(* PLC project steel-plant, Generated TextualNotationConverter 1.0 *)
(* stored: creationDateTime 2025-07-30T12:00:00, modificationDateTime 2025-01-30T12:00:00 *)

FUNCTION_BLOCK ANALOG_IN
  VAR_INPUT
    Name : STRING;
    Description : STRING;
    Raw_Signal : REAL;
    PV_High : REAL;
    PV_Low : REAL;
    Scaling_Slope : REAL;
    Scaling_Offset : REAL;
    Alarm_Enable : BOOL;
  END_VAR
  VAR_OUTPUT
    PV : REAL;
    High_Alarm : BOOL;
    Low_Alarm : BOOL;
    General_Fault : BOOL;
  END_VAR

            
          
END_FUNCTION_BLOCK

FUNCTION_BLOCK PID_BASIC
  VAR_INPUT
    Name : STRING;
    Description : STRING;
    AUTO : BOOL;
    PV : REAL;
    SP : REAL;
    MV_MIN : REAL;
    MV_MAX : REAL;
    X0 : REAL;
    KP : REAL;
    TR : REAL;
    TD : REAL;
    PV_High : REAL;
    PV_Low : REAL;
    Deviation_Limit : REAL;
    Inhibit : BOOL;
  END_VAR
  VAR_OUTPUT
    PV_High_Alarm : BOOL;
    PV_Low_Alarm : BOOL;
    Deviation_Alarm : BOOL;
    XOUT : REAL;
  END_VAR

            
          
END_FUNCTION_BLOCK

FUNCTION_BLOCK RATIO_CONTROL
  VAR_INPUT
    Name : STRING;
    Description : STRING;
    Auto : BOOL;
    PrimaryPV : REAL;
    SecondaryPV : REAL;
    RatioSP : REAL;
    Bias : REAL;
    TrimKp : REAL;
    TrimTi : STRING;
    MV_MIN : REAL;
    MV_MAX : REAL;
    ManOut : REAL;
    Inhibit : BOOL;
  END_VAR
  VAR_OUTPUT
    SlaveSP : REAL;
    ActiveRatio : REAL;
    RatioErr : REAL;
  END_VAR

            
          
END_FUNCTION_BLOCK

FUNCTION_BLOCK VALVE_ELECTRIC
  VAR_INPUT
    Name : STRING;
    Description : STRING;
    Control_Signal : REAL;
    Manual_Mode : BOOL;
    Manual_Position : REAL;
    Open_Limit : REAL;
    Close_Limit : REAL;
    Timeout : STRING;
    Inhibit : BOOL;
  END_VAR
  VAR_OUTPUT
    Valve_Position : REAL;
    Feedback_Pos : REAL;
    Valve_Moving : BOOL;
    Position_Error : BOOL;
    Alarm : BOOL;
  END_VAR

            
          
END_FUNCTION_BLOCK

PROGRAM Section2
  VAR
    FT101_WildFlow_PV : REAL;
    FT102_FluxFlow_PV : REAL;
    TIT101_Temperature_PV : REAL;
    FFIC103_FluxFlow_SP : REAL;
  END_VAR
  VAR
    FT-101 : ANALOG_IN;
    FT-102 : ANALOG_IN;
    TIT-101 : ANALOG_IN;
    FFIC-103 : RATIO_CONTROL;
    FIC-102 : PID_BASIC;
    FV-102 : VALVE_ELECTRIC;
  END_VAR
  VAR  (* added by the conversion: wires and edge detectors of the diagram *)
    _GT1_OUT : BOOL;
    _OR2_OUT : BOOL;
  END_VAR

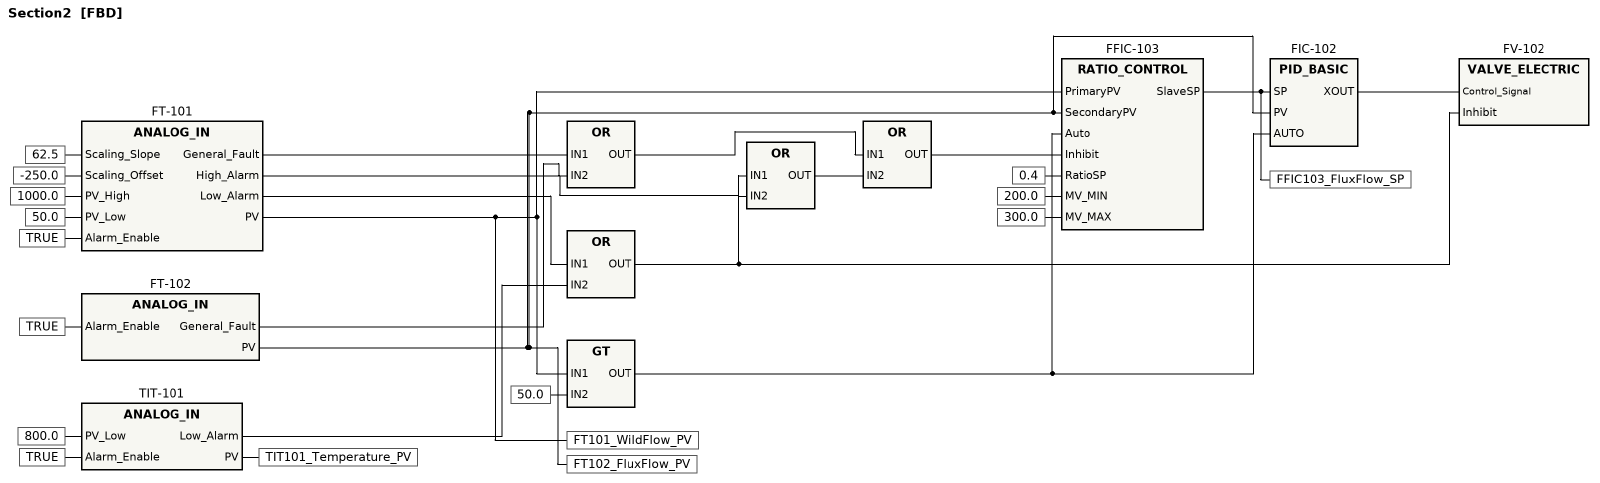
(* FBD diagram, written out as Structured Text *)
FT-101(Scaling_Slope := 62.5, Scaling_Offset := -250.0, PV_High := 1000.0, PV_Low := 50.0, Alarm_Enable := TRUE);
FT-102(Alarm_Enable := TRUE);
_GT1_OUT := FT-101.PV > 50.0;
TIT-101(PV_Low := 800.0, Alarm_Enable := TRUE);
_OR2_OUT := FT-101.Low_Alarm OR TIT-101.Low_Alarm;
FFIC-103(PrimaryPV := FT-101.PV, SecondaryPV := FT-102.PV, Auto := _GT1_OUT, Inhibit := FT-101.General_Fault OR FT-102.General_Fault OR FT-101.High_Alarm OR _OR2_OUT, RatioSP := 0.4, MV_MIN := 200.0, MV_MAX := 300.0);
FFIC103_FluxFlow_SP := FFIC-103.SlaveSP;
FT101_WildFlow_PV := FT-101.PV;
FT102_FluxFlow_PV := FT-102.PV;
TIT101_Temperature_PV := TIT-101.PV;
FIC-102(SP := FFIC-103.SlaveSP, PV := FT-102.PV, AUTO := _GT1_OUT);
FV-102(Control_Signal := FIC-102.XOUT, Inhibit := _OR2_OUT);
END_PROGRAM

FUNCTION_BLOCK BOOL_IN
  VAR_INPUT
    Name : STRING;
    Description : STRING;
    Bool_In : BOOL;
    Alarm_OnTrue : BOOL;
    Alarm_OnFalse : BOOL;
    Latch_Enable : BOOL;
    Reset_Latch : BOOL;
  END_VAR
  VAR_OUTPUT
    Bool_Out : BOOL;
    Alarm_Active : BOOL;
    Latched_Status : BOOL;
  END_VAR

            
          
END_FUNCTION_BLOCK

FUNCTION_BLOCK DIGITAL_IN
  VAR_INPUT
    Name : STRING;
    Description : STRING;
    DI_Raw : BOOL;
    DebounceTime : STRING;
    EnableAlarm : BOOL;
  END_VAR
  VAR_OUTPUT
    DI_Out : BOOL;
    Fault_State : BOOL;
  END_VAR

            
          
END_FUNCTION_BLOCK

FUNCTION_BLOCK DUTY_STANDBY
  VAR_INPUT
    Name : STRING;
    Description : STRING;
    Enable : BOOL;
    StartRequest : BOOL;
    AlternateEnable : BOOL;
    ForcePumpA : BOOL;
    ForcePumpB : BOOL;
    DutyElapsed : BOOL;
    MinRunElapsed : BOOL;
    SwitchoverDelayElapsed : BOOL;
    StartTimeoutElapsed : BOOL;
    PumpA_RunFB : BOOL;
    PumpB_RunFB : BOOL;
    PumpA_Fault : BOOL;
    PumpB_Fault : BOOL;
    Reset : BOOL;
    Inhibit : BOOL;
  END_VAR
  VAR_OUTPUT
    CmdPumpA : BOOL;
    CmdPumpB : BOOL;
    ActiveIsA : BOOL;
    SwitchedDueToDuty : BOOL;
    SwitchedDueToFailure : BOOL;
    Alarm_FailedStart_A : BOOL;
    Alarm_FailedStart_B : BOOL;
    Alarm_NoAvailablePump : BOOL;
  END_VAR

            
          
END_FUNCTION_BLOCK

FUNCTION_BLOCK MOTOR_2SPD
  VAR_INPUT
    Name : STRING;
    Description : STRING;
    Start_Cmd : BOOL;
    Stop_Cmd : BOOL;
    Speed_High_Cmd : BOOL;
    Speed_Low_Cmd : BOOL;
    Inhibit : BOOL;
  END_VAR
  VAR_OUTPUT
    Motor_Start_Out : BOOL;
    FB_Running : BOOL;
    FB_Trip : BOOL;
    FB_HighSpeed : BOOL;
    FB_LowSpeed : BOOL;
    Alarm_Speed_Error : BOOL;
  END_VAR

            
          
END_FUNCTION_BLOCK

FUNCTION_BLOCK MOTOR_ON_OFF
  VAR_INPUT
    Name : STRING;
    Description : STRING;
    Start_Cmd : BOOL;
    Stop_Cmd : BOOL;
    Start_Delay : STRING;
    MinRunTime : STRING;
    Inhibit : BOOL;
  END_VAR
  VAR_OUTPUT
    Motor_Start_Out : BOOL;
    FB_Running : BOOL;
    FB_Trip : BOOL;
    Alarm_Start_Fail : BOOL;
    Alarm_Stop_Fail : BOOL;
  END_VAR

            
          
END_FUNCTION_BLOCK

FUNCTION_BLOCK MOTOR_VSD
  VAR_INPUT
    Name : STRING;
    Description : STRING;
    Start_Cmd : BOOL;
    Stop_Cmd : BOOL;
    Speed_SP : REAL;
    Accel_Ramp : STRING;
    Decel_Ramp : STRING;
    Inhibit : BOOL;
  END_VAR
  VAR_OUTPUT
    Speed_Out : REAL;
    FB_Running : BOOL;
    FB_Fault : BOOL;
    FB_Ready : BOOL;
    FB_ActualSpeed : REAL;
    Alarm_Speed_Deviation : BOOL;
    Alarm_Comm_Fail : BOOL;
  END_VAR

            
          
END_FUNCTION_BLOCK

FUNCTION_BLOCK SPLIT_RANGE
  VAR_INPUT
    Name : STRING;
    Description : STRING;
    IN : REAL;
    Split_Point : REAL;
    Output1_Start : REAL;
    Output1_End : REAL;
    Output2_Start : REAL;
    Output2_End : REAL;
  END_VAR
  VAR_OUTPUT
    OUT1 : REAL;
    OUT2 : REAL;
  END_VAR

            
          
END_FUNCTION_BLOCK

FUNCTION_BLOCK VALVE_ON_OFF
  VAR_INPUT
    Name : STRING;
    Description : STRING;
    Open_Cmd : BOOL;
    Close_Cmd : BOOL;
    Timeout : STRING;
    Inhibit : BOOL;
  END_VAR
  VAR_OUTPUT
    FB_Opened : BOOL;
    FB_Closed : BOOL;
    Valve_Open_Out : BOOL;
    Valve_Close_Out : BOOL;
    Alarm_Position_Error : BOOL;
    Alarm_General : BOOL;
  END_VAR

            
          
END_FUNCTION_BLOCK

FUNCTION_BLOCK VOTING_ANALOG
  VAR_INPUT
    Name : STRING;
    Description : STRING;
    Input1 : REAL;
    Input2 : REAL;
    Input3 : REAL;
    Deviation_Limit : REAL;
    Voting_Scheme : STRING;
    EnableAlarm : BOOL;
    Inhibit : BOOL;
  END_VAR
  VAR_OUTPUT
    Voted_Output : REAL;
    Sensor1_Fault : BOOL;
    Sensor2_Fault : BOOL;
    Sensor3_Fault : BOOL;
    Alarm_Voting_Error : BOOL;
    Healthy_Sensors_Count : INT;
  END_VAR

            
          
END_FUNCTION_BLOCK

PROGRAM Section3
  VAR
    PT_201_VOTE_PV : REAL;
    TT_201_VOTE_PV : REAL;
  END_VAR
  VAR
    PT-201A : ANALOG_IN;
    PT-201B : ANALOG_IN;
    PT-201C : ANALOG_IN;
    TT-201A : ANALOG_IN;
    TT-201B : ANALOG_IN;
    TT-201C : ANALOG_IN;
    PT-201_VOTE : VOTING_ANALOG;
    TT-201_VOTE : VOTING_ANALOG;
    P-201 : MOTOR_ON_OFF;
    MO-201 : DIGITAL_IN;
    MO-202 : DIGITAL_IN;
    I-201 : BOOL_IN;
    I-202 : BOOL_IN;
    SI-201 : BOOL_IN;
    SI-202 : BOOL_IN;
  END_VAR
  VAR  (* added by the conversion: wires and edge detectors of the diagram *)
    _OR37_OUT : BOOL;
  END_VAR

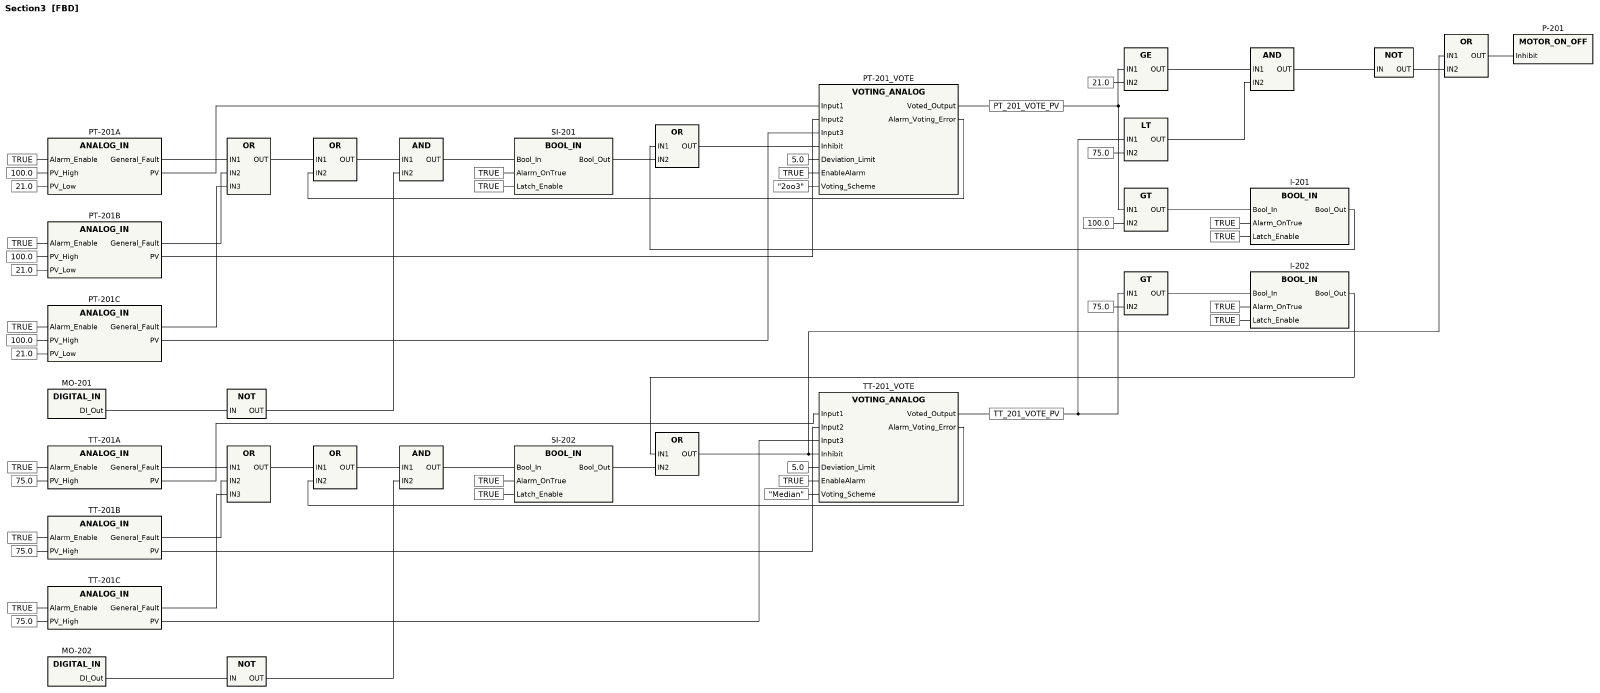
(* FBD diagram, written out as Structured Text *)
PT-201A(Alarm_Enable := TRUE, PV_High := 100.0, PV_Low := 21.0);
PT-201B(Alarm_Enable := TRUE, PV_High := 100.0, PV_Low := 21.0);
PT-201C(Alarm_Enable := TRUE, PV_High := 100.0, PV_Low := 21.0);
I-201(Bool_In := PT-201_VOTE.Voted_Output > 100.0, Alarm_OnTrue := TRUE, Latch_Enable := TRUE);
MO-201();
SI-201(Bool_In := (PT-201A.General_Fault OR PT-201B.General_Fault OR PT-201C.General_Fault OR PT-201_VOTE.Alarm_Voting_Error) AND NOT MO-201.DI_Out, Alarm_OnTrue := TRUE, Latch_Enable := TRUE);
PT-201_VOTE(Input1 := PT-201A.PV, Input2 := PT-201B.PV, Input3 := PT-201C.PV, Inhibit := I-201.Bool_Out OR SI-201.Bool_Out, Deviation_Limit := 5.0, EnableAlarm := TRUE, Voting_Scheme := "2oo3");
PT_201_VOTE_PV := PT-201_VOTE.Voted_Output;
TT-201A(Alarm_Enable := TRUE, PV_High := 75.0);
TT-201B(Alarm_Enable := TRUE, PV_High := 75.0);
TT-201C(Alarm_Enable := TRUE, PV_High := 75.0);
I-202(Bool_In := TT-201_VOTE.Voted_Output > 75.0, Alarm_OnTrue := TRUE, Latch_Enable := TRUE);
MO-202();
SI-202(Bool_In := (TT-201A.General_Fault OR TT-201B.General_Fault OR TT-201C.General_Fault OR TT-201_VOTE.Alarm_Voting_Error) AND NOT MO-202.DI_Out, Alarm_OnTrue := TRUE, Latch_Enable := TRUE);
_OR37_OUT := I-202.Bool_Out OR SI-202.Bool_Out;
TT-201_VOTE(Input1 := TT-201A.PV, Input2 := TT-201B.PV, Input3 := TT-201C.PV, Inhibit := _OR37_OUT, Deviation_Limit := 5.0, EnableAlarm := TRUE, Voting_Scheme := "Median");
TT_201_VOTE_PV := TT-201_VOTE.Voted_Output;
P-201(Inhibit := _OR37_OUT OR NOT (PT-201_VOTE.Voted_Output >= 21.0 AND TT-201_VOTE.Voted_Output < 75.0));
END_PROGRAM

PROGRAM Section4
  VAR
    FT_301_CoalFlow_PV : REAL;
    FT_302_AirFlow_PV : REAL;
    PT_301_Pressure_PV : REAL;
    TT_301_Temperature_PV : REAL;
    FIC_302_HotBlastAir_SP_FromRatio : REAL;
    Ratio_Bias : REAL;
  END_VAR
  VAR
    FT-301 : ANALOG_IN;
    PT-301 : ANALOG_IN;
    TT-301 : ANALOG_IN;
    FT-302 : ANALOG_IN;
    FFIC-303 : RATIO_CONTROL;
    FIC-302 : PID_BASIC;
    FV-302 : VALVE_ELECTRIC;
  END_VAR
  VAR  (* added by the conversion: wires and edge detectors of the diagram *)
    _OR95_OUT : BOOL;
    _OR96_OUT : BOOL;
  END_VAR

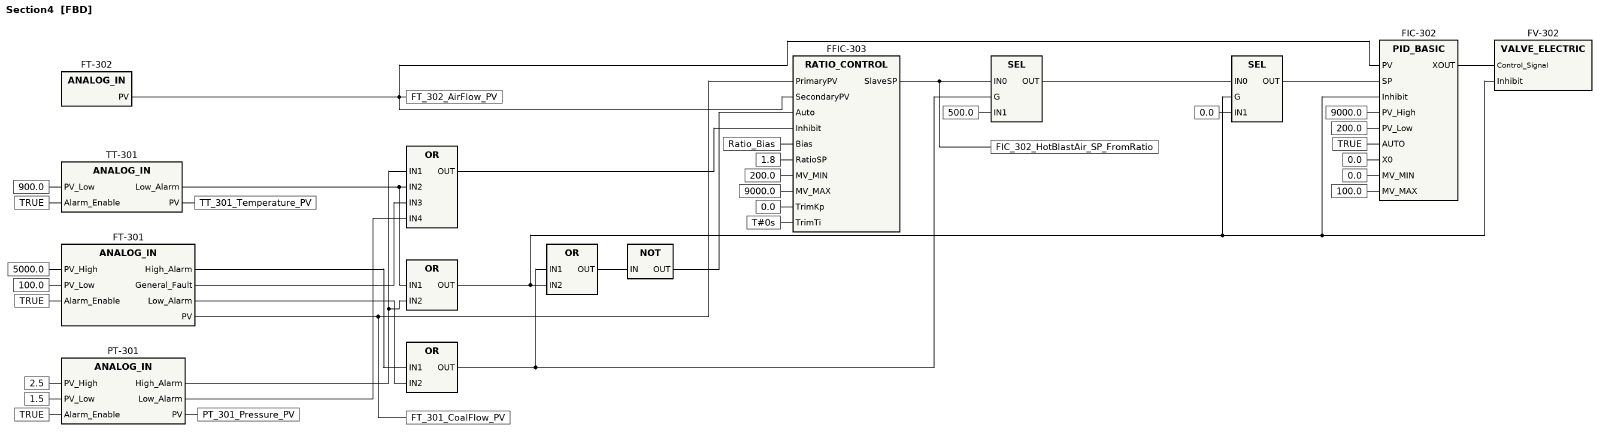
(* FBD diagram, written out as Structured Text *)
FT-301(PV_High := 5000.0, PV_Low := 100.0, Alarm_Enable := TRUE);
FT-302();
_OR95_OUT := FT-301.High_Alarm OR FT-301.Low_Alarm;
TT-301(PV_Low := 900.0, Alarm_Enable := TRUE);
PT-301(PV_High := 2.5, PV_Low := 1.5, Alarm_Enable := TRUE);
_OR96_OUT := TT-301.Low_Alarm OR PT-301.High_Alarm;
FFIC-303(PrimaryPV := FT-301.PV, SecondaryPV := FT-302.PV, Auto := NOT (_OR95_OUT OR _OR96_OUT), Inhibit := PT-301.High_Alarm OR TT-301.Low_Alarm OR FT-301.General_Fault OR PT-301.Low_Alarm, Bias := Ratio_Bias, RatioSP := 1.8, MV_MIN := 200.0, MV_MAX := 9000.0, TrimKp := 0.0, TrimTi := T#0s);
FIC_302_HotBlastAir_SP_FromRatio := FFIC-303.SlaveSP;
FT_301_CoalFlow_PV := FT-301.PV;
FT_302_AirFlow_PV := FT-302.PV;
PT_301_Pressure_PV := PT-301.PV;
TT_301_Temperature_PV := TT-301.PV;
FIC-302(PV := FT-302.PV, SP := SEL(SEL(FFIC-303.SlaveSP, _OR95_OUT, 500.0), _OR96_OUT, 0.0), Inhibit := _OR96_OUT, PV_High := 9000.0, PV_Low := 200.0, AUTO := TRUE, X0 := 0.0, MV_MIN := 0.0, MV_MAX := 100.0);
FV-302(Control_Signal := FIC-302.XOUT, Inhibit := _OR96_OUT);
END_PROGRAM

PROGRAM Section5
  VAR
    TT_401_V_Temp_PV : REAL;
    PT_401_V_Pressure_PV : REAL;
    FT_401_Flow_PV : REAL;
  END_VAR
  VAR
    FT-401 : ANALOG_IN;
    PT-401A : ANALOG_IN;
    PT-401B : ANALOG_IN;
    PT-401C : ANALOG_IN;
    TT-401 : ANALOG_IN;
    TT-401A : ANALOG_IN;
    TT-401B : ANALOG_IN;
    TT-401C : ANALOG_IN;
    TT-401-V : VOTING_ANALOG;
    PT-401-V : VOTING_ANALOG;
    BOF-401_TempControl : PID_BASIC;
    BOF-402 : VALVE_ELECTRIC;
    I-401 : BOOL_IN;
    MA-401 : BOOL_IN;
    DA-401 : BOOL_IN;
    FA-401 : BOOL_IN;
  END_VAR
  VAR  (* added by the conversion: wires and edge detectors of the diagram *)
    _AND143_OUT : BOOL;
    _AND144_OUT : BOOL;
    _AND145_OUT : BOOL;
  END_VAR

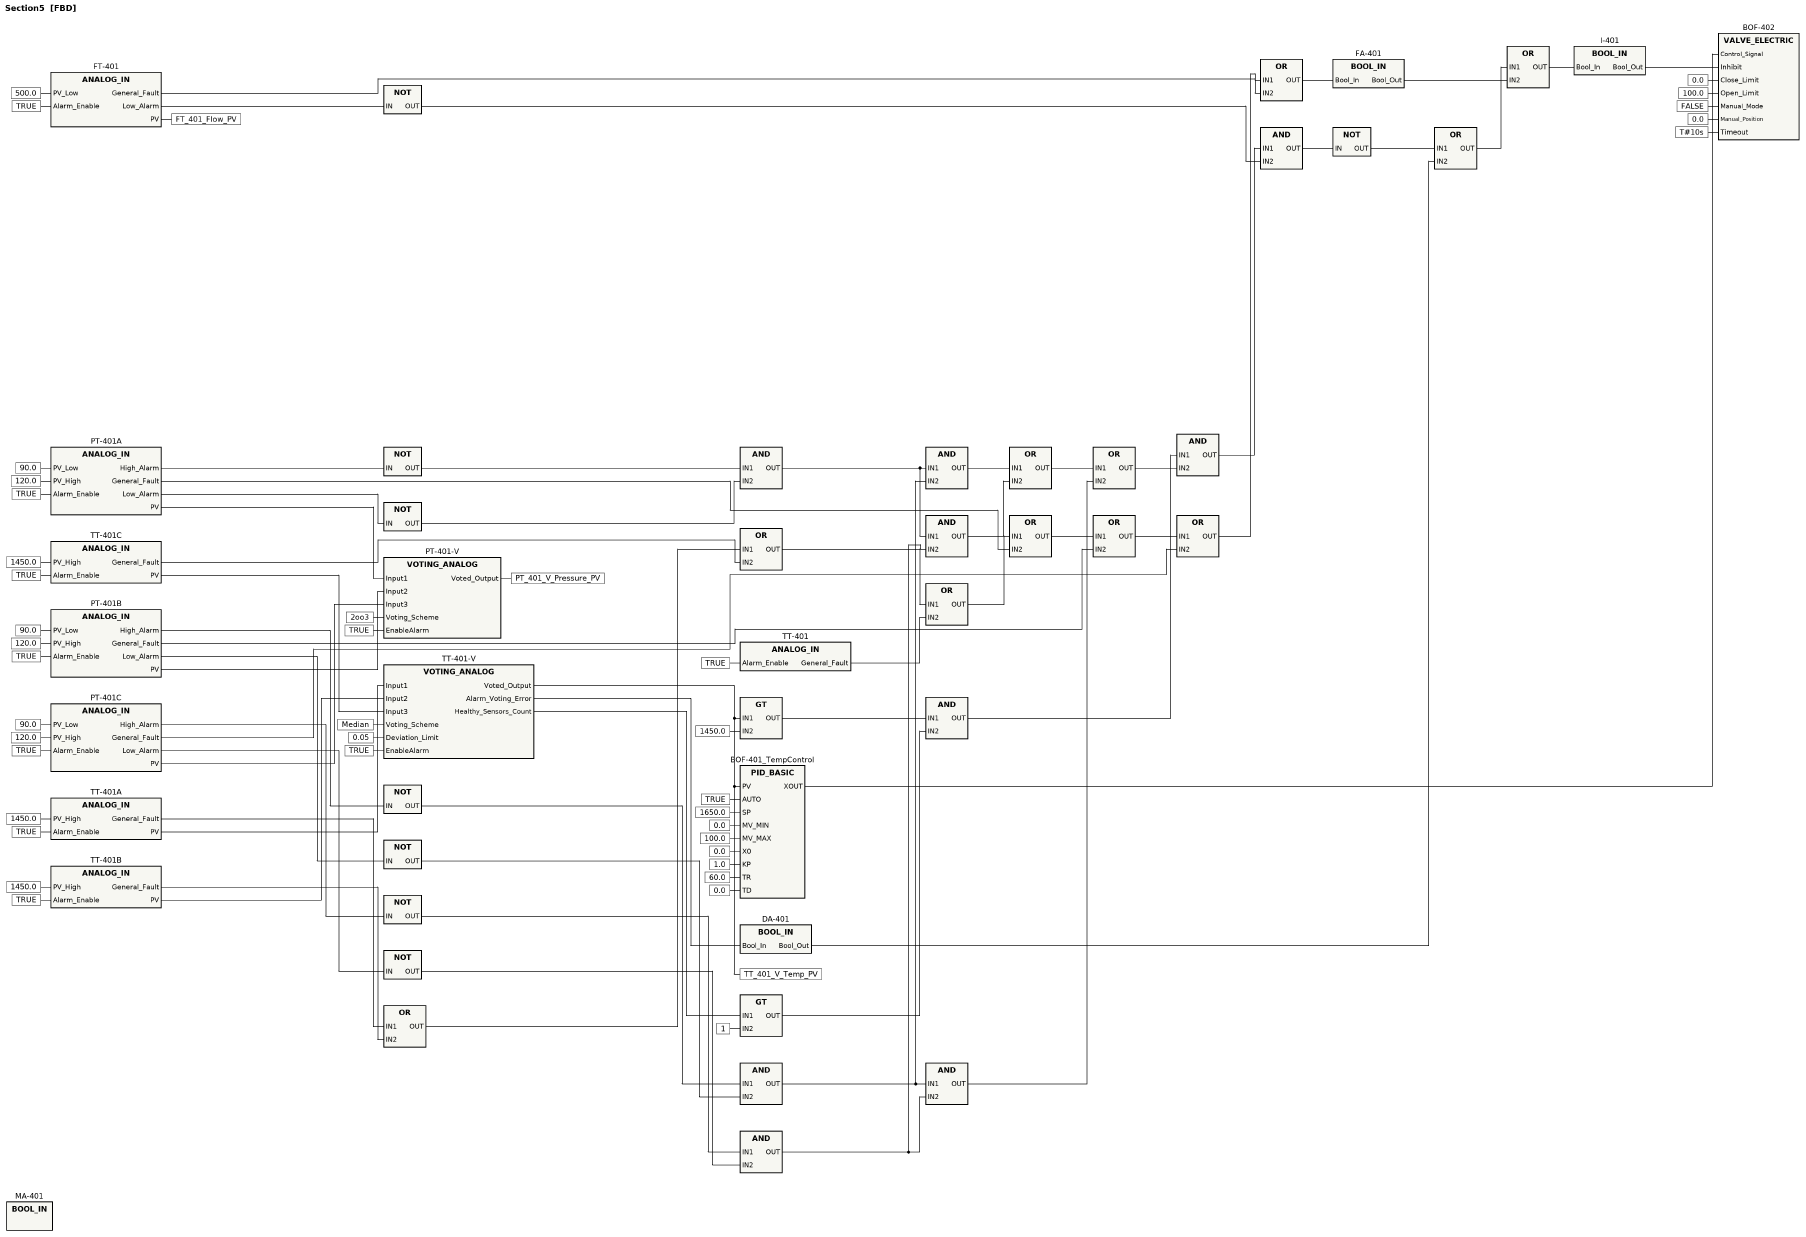
(* FBD diagram, written out as Structured Text *)
FT-401(PV_Low := 500.0, Alarm_Enable := TRUE);
FT_401_Flow_PV := FT-401.PV;
PT-401A(PV_Low := 90.0, PV_High := 120.0, Alarm_Enable := TRUE);
PT-401B(PV_Low := 90.0, PV_High := 120.0, Alarm_Enable := TRUE);
PT-401C(PV_Low := 90.0, PV_High := 120.0, Alarm_Enable := TRUE);
PT-401-V(Input1 := PT-401A.PV, Input2 := PT-401B.PV, Input3 := PT-401C.PV, Voting_Scheme := 2oo3, EnableAlarm := TRUE);
PT_401_V_Pressure_PV := PT-401-V.Voted_Output;
TT-401A(PV_High := 1450.0, Alarm_Enable := TRUE);
TT-401B(PV_High := 1450.0, Alarm_Enable := TRUE);
TT-401C(PV_High := 1450.0, Alarm_Enable := TRUE);
TT-401-V(Input1 := TT-401A.PV, Input2 := TT-401B.PV, Input3 := TT-401C.PV, Voting_Scheme := Median, Deviation_Limit := 0.05, EnableAlarm := TRUE);
TT_401_V_Temp_PV := TT-401-V.Voted_Output;
_AND143_OUT := NOT PT-401A.High_Alarm AND NOT PT-401A.Low_Alarm;
_AND144_OUT := NOT PT-401B.High_Alarm AND NOT PT-401B.Low_Alarm;
_AND145_OUT := NOT PT-401C.High_Alarm AND NOT PT-401C.Low_Alarm;
TT-401(Alarm_Enable := TRUE);
DA-401(Bool_In := TT-401-V.Alarm_Voting_Error);
FA-401(Bool_In := TT-401A.General_Fault OR TT-401B.General_Fault OR TT-401C.General_Fault OR TT-401.General_Fault OR PT-401A.General_Fault OR PT-401B.General_Fault OR PT-401C.General_Fault OR FT-401.General_Fault);
BOF-401_TempControl(PV := TT-401-V.Voted_Output, AUTO := TRUE, SP := 1650.0, MV_MIN := 0.0, MV_MAX := 100.0, X0 := 0.0, KP := 1.0, TR := 60.0, TD := 0.0);
I-401(Bool_In := NOT (TT-401-V.Voted_Output > 1450.0 AND TT-401-V.Healthy_Sensors_Count > 1 AND (_AND143_OUT AND _AND144_OUT OR _AND143_OUT AND _AND145_OUT OR _AND144_OUT AND _AND145_OUT) AND NOT FT-401.Low_Alarm) OR DA-401.Bool_Out OR FA-401.Bool_Out);
BOF-402(Control_Signal := BOF-401_TempControl.XOUT, Inhibit := I-401.Bool_Out, Close_Limit := 0.0, Open_Limit := 100.0, Manual_Mode := FALSE, Manual_Position := 0.0, Timeout := T#10s);
MA-401();
END_PROGRAM

PROGRAM Section6
  VAR
    PT_501_Pressure_PV : REAL;
    TT_501_Temperature_PV : REAL;
    TT_501_MV : REAL;
    SM_501_EA_POS : REAL;
    SM_501_EA_CMD : REAL;
  END_VAR
  VAR
    PT-501 : ANALOG_IN;
    TT-501 : ANALOG_IN;
    SM-501 : VALVE_ELECTRIC;
    TT-501_CTRL : PID_BASIC;
    SM-501.LID_POS : DIGITAL_IN;
    HeatingEnableDelay_TON : TON;
  END_VAR
  VAR  (* added by the conversion: wires and edge detectors of the diagram *)
    _OR223_OUT : BOOL;
  END_VAR

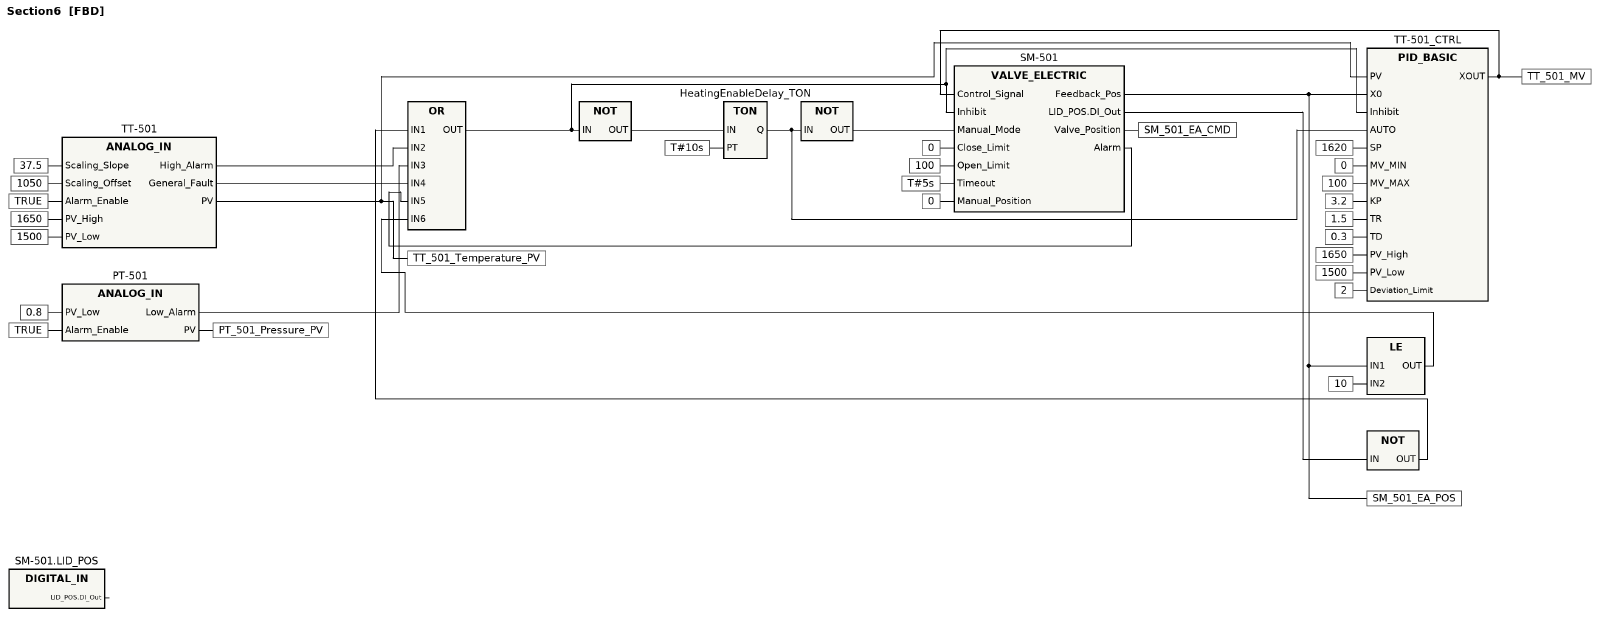
(* FBD diagram, written out as Structured Text *)
PT-501(PV_Low := 0.8, Alarm_Enable := TRUE);
PT_501_Pressure_PV := PT-501.PV;
TT-501(Scaling_Slope := 37.5, Scaling_Offset := 1050, Alarm_Enable := TRUE, PV_High := 1650, PV_Low := 1500);
_OR223_OUT := NOT SM-501.LID_POS.DI_Out OR TT-501.High_Alarm OR PT-501.Low_Alarm OR TT-501.General_Fault OR SM-501.Alarm OR SM-501.Feedback_Pos <= 10;
HeatingEnableDelay_TON(IN := NOT _OR223_OUT, PT := T#10s);
TT-501_CTRL(PV := TT-501.PV, X0 := SM-501.Feedback_Pos, Inhibit := _OR223_OUT, AUTO := HeatingEnableDelay_TON.Q, SP := 1620, MV_MIN := 0, MV_MAX := 100, KP := 3.2, TR := 1.5, TD := 0.3, PV_High := 1650, PV_Low := 1500, Deviation_Limit := 2);
SM-501(Control_Signal := TT-501_CTRL.XOUT, Inhibit := _OR223_OUT, Manual_Mode := NOT HeatingEnableDelay_TON.Q, Close_Limit := 0, Open_Limit := 100, Timeout := T#5s, Manual_Position := 0);
SM_501_EA_CMD := SM-501.Valve_Position;
SM_501_EA_POS := SM-501.Feedback_Pos;
TT_501_MV := TT-501_CTRL.XOUT;
TT_501_Temperature_PV := TT-501.PV;
SM-501.LID_POS();
END_PROGRAM

PROGRAM Section7
  VAR
    LIT101_MoldLevel_PV_mm : REAL;
    FT601_CoolingWaterFlow_PV_m3h : REAL;
    TT601_MoldTemp_PV_C : REAL;
    LIC101_ControllerOutput_Pct : REAL;
  END_VAR
  VAR
    LIT-101 : ANALOG_IN;
    FT-601 : ANALOG_IN;
    TT-601 : ANALOG_IN;
    LIC-101 : PID_BASIC;
    MV-101 : VALVE_ELECTRIC;
    ILK-FT-601-LOW : BOOL_IN;
    ILK-TT-601-HIGH : BOOL_IN;
    PERM-LIT-101-UNDER-250 : BOOL_IN;
    ILK-LIT-101-HIGH-HIGH-280 : BOOL_IN;
    ILK-LIT-101-FAULT : BOOL_IN;
  END_VAR
  VAR  (* added by the conversion: wires and edge detectors of the diagram *)
    _OR261_OUT : BOOL;
  END_VAR

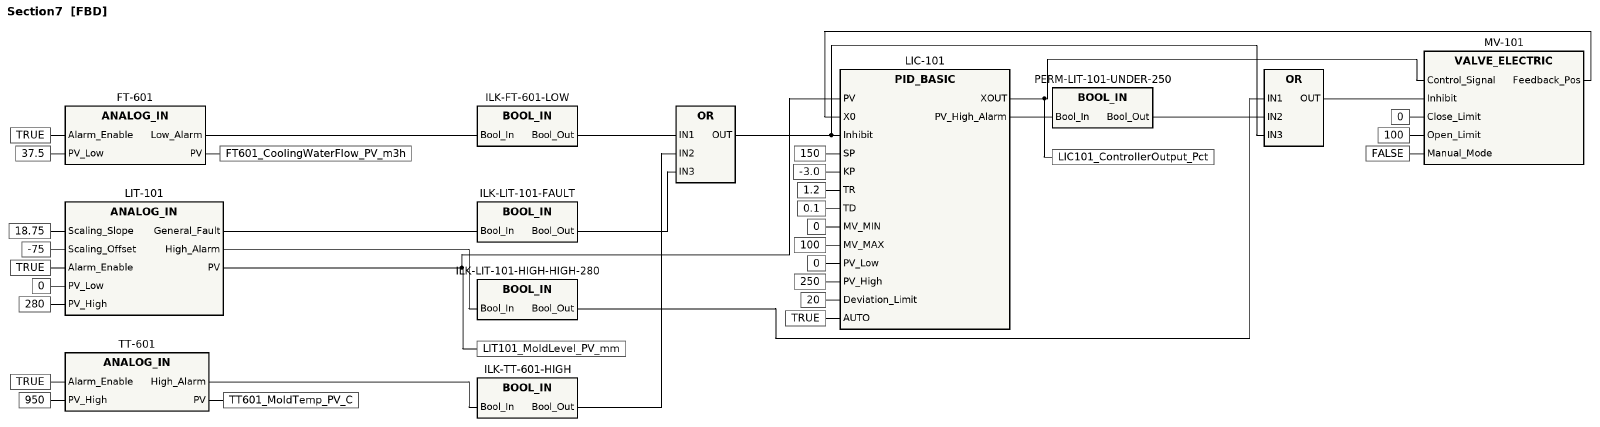
(* FBD diagram, written out as Structured Text *)
FT-601(Alarm_Enable := TRUE, PV_Low := 37.5);
FT601_CoolingWaterFlow_PV_m3h := FT-601.PV;
LIT-101(Scaling_Slope := 18.75, Scaling_Offset := -75, Alarm_Enable := TRUE, PV_Low := 0, PV_High := 280);
ILK-LIT-101-HIGH-HIGH-280(Bool_In := LIT-101.High_Alarm);
PERM-LIT-101-UNDER-250(Bool_In := LIC-101.PV_High_Alarm);
ILK-FT-601-LOW(Bool_In := FT-601.Low_Alarm);
TT-601(Alarm_Enable := TRUE, PV_High := 950);
ILK-TT-601-HIGH(Bool_In := TT-601.High_Alarm);
ILK-LIT-101-FAULT(Bool_In := LIT-101.General_Fault);
_OR261_OUT := ILK-FT-601-LOW.Bool_Out OR ILK-TT-601-HIGH.Bool_Out OR ILK-LIT-101-FAULT.Bool_Out;
MV-101(Control_Signal := LIC-101.XOUT, Inhibit := ILK-LIT-101-HIGH-HIGH-280.Bool_Out OR PERM-LIT-101-UNDER-250.Bool_Out OR _OR261_OUT, Close_Limit := 0, Open_Limit := 100, Manual_Mode := FALSE);
LIC-101(PV := LIT-101.PV, X0 := MV-101.Feedback_Pos, Inhibit := _OR261_OUT, SP := 150, KP := -3.0, TR := 1.2, TD := 0.1, MV_MIN := 0, MV_MAX := 100, PV_Low := 0, PV_High := 250, Deviation_Limit := 20, AUTO := TRUE);
LIC101_ControllerOutput_Pct := LIC-101.XOUT;
LIT101_MoldLevel_PV_mm := LIT-101.PV;
TT601_MoldTemp_PV_C := TT-601.PV;
END_PROGRAM

PROGRAM Section8
  VAR
    FT701_FuelFlow_PV : REAL;
    FT702_AirFlow_PV : REAL;
    TT701_FurnaceTemp_PV : REAL;
    FLT701_FuelTankLevel_PV : REAL;
    FT702_SP_Ratio : REAL;
    FFIC701_ActiveRatio : REAL;
    FFIC701_RatioError : REAL;
    BLS701_BurnerStatus : BOOL;
    BLS701_BurnerStatus_DI : BOOL;
    ALM701_RatioAlarm : BOOL;
    ALM702_FT701Fault : BOOL;
    ALM703_FT702Fault : BOOL;
    ALM704_HighTemp : BOOL;
  END_VAR
  VAR
    FT-701 : ANALOG_IN;
    FT-702 : ANALOG_IN;
    TT-701 : ANALOG_IN;
    FLT-701 : ANALOG_IN;
    FFIC-701 : RATIO_CONTROL;
    FIC-702 : PID_BASIC;
    FV-702 : VALVE_ELECTRIC;
    BLS-701 : BOOL_IN;
  END_VAR
  VAR  (* added by the conversion: wires and edge detectors of the diagram *)
    _NOT300_OUT : BOOL;
    _OR301_OUT : BOOL;
  END_VAR

(* FBD diagram, written out as Structured Text *)
FT-701(PV_High := 5000.0, PV_Low := 200.0, Alarm_Enable := TRUE);
FT-702(PV_High := 15000.0, PV_Low := 0.0, Alarm_Enable := TRUE);
TT-701(PV_High := 1200.0, PV_Low := 800.0, Alarm_Enable := TRUE);
BLS-701(Bool_In := BLS701_BurnerStatus_DI, Alarm_OnFalse := TRUE, Alarm_OnTrue := FALSE, Latch_Enable := FALSE);
_NOT300_OUT := NOT BLS-701.Bool_Out;
_OR301_OUT := FT-701.General_Fault OR FT-702.General_Fault;
FFIC-701(PrimaryPV := FT-701.PV, SecondaryPV := FT-702.PV, Auto := NOT TT-701.High_Alarm AND FT-701.PV >= 200.0 AND BLS-701.Bool_Out, Inhibit := _NOT300_OUT OR FT-701.Low_Alarm OR _OR301_OUT, MV_MIN := MULT(FT-701.PV, 8.0), MV_MAX := MULT(FT-701.PV, 12.0), ManOut := MULT(FT-701.PV, 8.0), RatioSP := 10.0, Bias := 0.0);
ALM701_RatioAlarm := FFIC-701.ActiveRatio > 8.0 OR FFIC-701.ActiveRatio > 12.0;
ALM702_FT701Fault := FT-701.General_Fault;
ALM703_FT702Fault := FT-702.General_Fault;
ALM704_HighTemp := TT-701.High_Alarm;
BLS701_BurnerStatus := BLS-701.Bool_Out;
FFIC701_ActiveRatio := FFIC-701.ActiveRatio;
FFIC701_RatioError := FFIC-701.RatioErr;
FLT-701();
FLT701_FuelTankLevel_PV := FLT-701.PV;
FT701_FuelFlow_PV := FT-701.PV;
FT702_AirFlow_PV := FT-702.PV;
FT702_SP_Ratio := FFIC-701.SlaveSP;
TT701_FurnaceTemp_PV := TT-701.PV;
FIC-702(SP := FFIC-701.SlaveSP, PV := FT-702.PV, Inhibit := _NOT300_OUT OR _OR301_OUT, AUTO := TRUE, MV_MIN := 0.0, MV_MAX := 100.0, PV_High := 15000.0, PV_Low := 0.0, KP := 1.5, TR := 10.0, TD := 0.5, Deviation_Limit := 5.0, X0 := 0.0);
FV-702(Control_Signal := FIC-702.XOUT, Inhibit := FT-701.Low_Alarm OR TT-701.Low_Alarm OR TT-701.High_Alarm OR _OR301_OUT, Manual_Mode := FALSE, Close_Limit := 0.0, Open_Limit := 100.0, Timeout := T#10s);
END_PROGRAM

PROGRAM Section9
  VAR
    FT801_Flow_PV : REAL;
    FT802_Flow_PV : REAL;
    PT801_Pressure_PV : REAL;
    FFIC801_AirFlow_SP : REAL;
    FFIC801_ActiveRatio : REAL;
    RatioHigh_Alarm : BOOL;
    RatioLow_Alarm : BOOL;
  END_VAR
  VAR
    AL-801 : ANALOG_IN;
    AL-802 : ANALOG_IN;
    AL-803 : ANALOG_IN;
    AL-804 : ANALOG_IN;
    FT-801 : ANALOG_IN;
    FT-802 : ANALOG_IN;
    PT-801 : ANALOG_IN;
    FFIC-801 : RATIO_CONTROL;
    FIC-802 : PID_BASIC;
    FV-802 : VALVE_ELECTRIC;
  END_VAR
  VAR  (* added by the conversion: wires and edge detectors of the diagram *)
    _GE372_OUT : BOOL;
    _OR373_OUT : BOOL;
    _OR375_OUT : BOOL;
  END_VAR

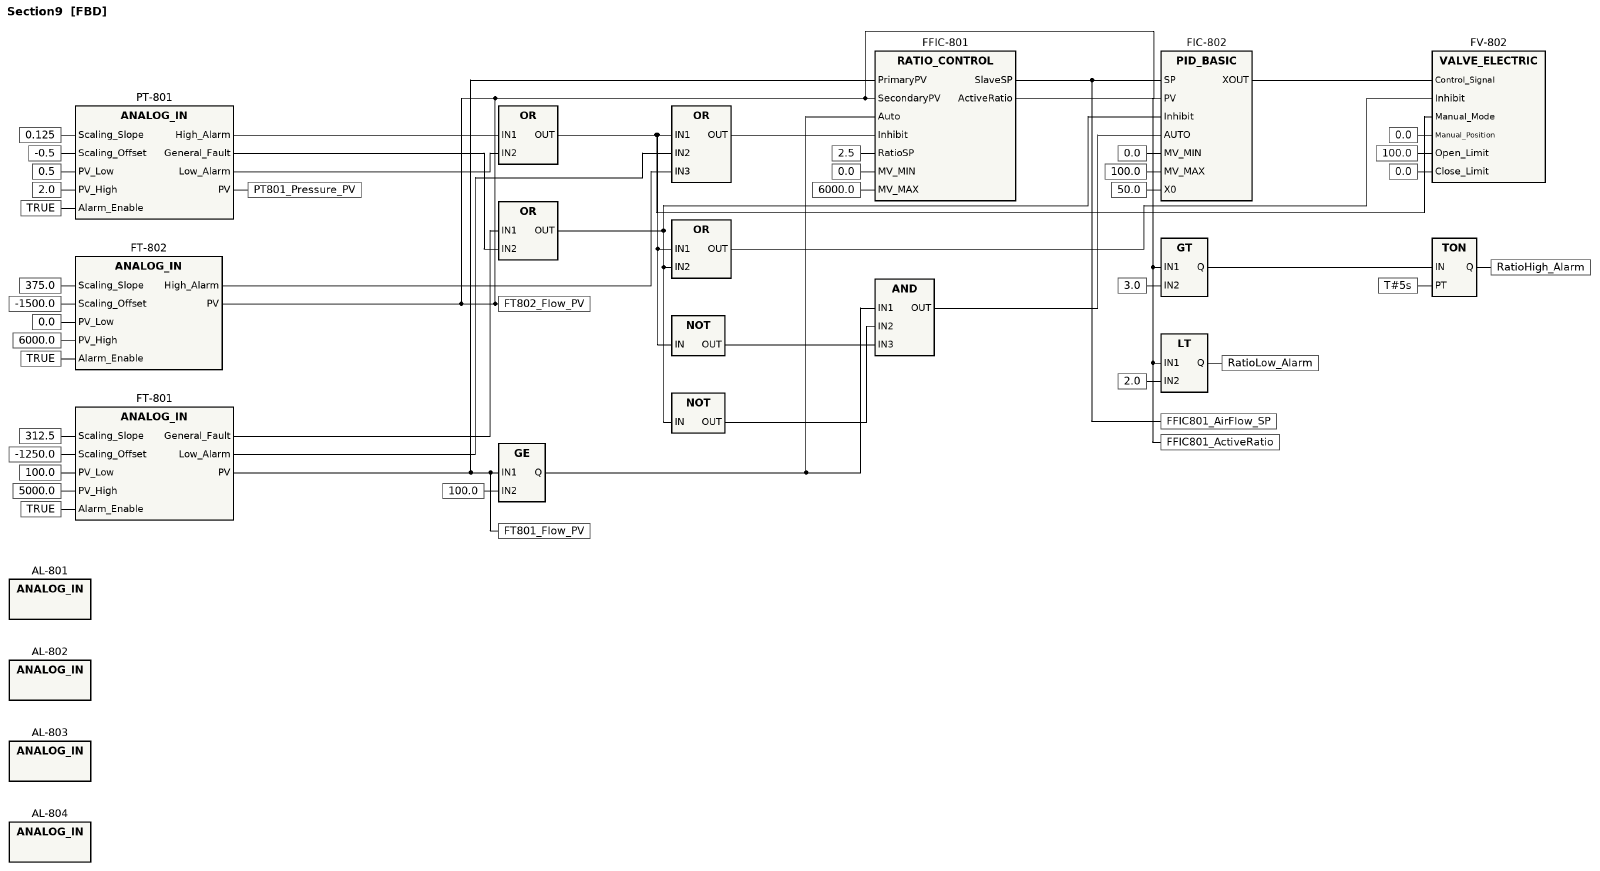
(* FBD diagram, written out as Structured Text *)
FT-801(Scaling_Slope := 312.5, Scaling_Offset := -1250.0, PV_Low := 100.0, PV_High := 5000.0, Alarm_Enable := TRUE);
FT-802(Scaling_Slope := 375.0, Scaling_Offset := -1500.0, PV_Low := 0.0, PV_High := 6000.0, Alarm_Enable := TRUE);
_GE372_OUT := FT-801.PV >= 100.0;
PT-801(Scaling_Slope := 0.125, Scaling_Offset := -0.5, PV_Low := 0.5, PV_High := 2.0, Alarm_Enable := TRUE);
_OR373_OUT := PT-801.High_Alarm OR PT-801.Low_Alarm;
FFIC-801(PrimaryPV := FT-801.PV, SecondaryPV := FT-802.PV, Auto := _GE372_OUT, Inhibit := _OR373_OUT OR FT-801.Low_Alarm OR FT-802.High_Alarm, RatioSP := 2.5, MV_MIN := 0.0, MV_MAX := 6000.0);
FFIC801_ActiveRatio := FFIC-801.ActiveRatio;
FFIC801_AirFlow_SP := FFIC-801.SlaveSP;
FT801_Flow_PV := FT-801.PV;
FT802_Flow_PV := FT-802.PV;
PT801_Pressure_PV := PT-801.PV;
RatioHigh_Alarm := TON(FFIC-801.ActiveRatio > 3.0, T#5s);
RatioLow_Alarm := FFIC-801.ActiveRatio < 2.0;
_OR375_OUT := FT-801.General_Fault OR PT-801.General_Fault;
AL-801();
AL-802();
AL-803();
AL-804();
FIC-802(SP := FFIC-801.SlaveSP, PV := FT-802.PV, Inhibit := _OR375_OUT, AUTO := _GE372_OUT AND NOT _OR375_OUT AND NOT _OR373_OUT, MV_MIN := 0.0, MV_MAX := 100.0, X0 := 50.0);
FV-802(Control_Signal := FIC-802.XOUT, Inhibit := _OR373_OUT OR _OR375_OUT, Manual_Mode := _OR373_OUT, Manual_Position := 0.0, Open_Limit := 100.0, Close_Limit := 0.0);
END_PROGRAM

CONFIGURATION Config0
  RESOURCE Res0 ON PLC
    TASK task0(INTERVAL := T#20ms, PRIORITY := 0);
    PROGRAM instance0 WITH task0 : Section2;
    PROGRAM instance_1 WITH task0 : Section3;
    PROGRAM instance_2 WITH task0 : Section4;
    PROGRAM instance_3 WITH task0 : Section5;
    PROGRAM instance_4 WITH task0 : Section6;
    PROGRAM instance_5 WITH task0 : Section7;
    PROGRAM instance_6 WITH task0 : Section8;
    PROGRAM instance_7 WITH task0 : Section9;
  END_RESOURCE
END_CONFIGURATION
